FUNCTION_BLOCK CalibrationBlock
VAR_INPUT

	fbMotorReference : REFERENCE TO FB_AnalogMotorDriver; 	

END_VAR
VAR_OUTPUT

	// Variables for logging 
	nEncoder1Counts : LINT; 
	rEncoder1Degrees : REAL; 	
	
	// Variables for motor control 
	rCommand : REAL; 
	
	// Variables for load cell 
	rGripForce : REAL; 

END_VAR

// Constants used for the program 
VAR CONSTANT
	nMaxTrialNumber : UINT := 10; 
END_VAR

VAR
	
	// Variables to keep track of the actual encoder/motor setup
	fbEncoder1 : FB_QuadratureEncoder; 
	fbLoadCell : FB_AnalogLoadCellInput; // TODO: Change everything to top level reference maybe? 
	
	////// BEGIN GUI TEST OPTIONS
	//// All fields in the next section are in some way or another set by the GUI, and define 
	//// the type of test to take place.
	// 1. Test type
	bTestTypeHuman : BOOL; // Whether or not this a human or motor test 
	bTestTypeHumanLIVE : BOOL; 
	
	// 2. Number of trials
	nTrialNumber : UINT := 1; // Number of calibration trials to run in succession 
	nTrialNumberLIVE : UINT; 
	
	// 3. Trigger type
	bManualPulse : BOOL; // Whether to use manual pulse or grip schedule. 
	bManualPulseLIVE : BOOL; 
	bManualPulseTimerEnable : BOOL; 
	bManualPulseTimerEnableLIVE : BOOL;
	rManualPulseTimerValue : REAL; 
	rManualPulseTimerValueLIVE : REAL;
	
	// 4. Trigger controls
	bUseConstantGripTrigger : BOOL;
	bUseConstantGripTriggerLIVE : BOOL;
	aGripSchedule : ARRAY[1..nMaxTrialNumber] OF REAL;
	aGripScheduleLIVE : ARRAY[1..nMaxTrialNumber] OF REAL;  
	rCurrentGripThreshold : REAL := 0; 
	
	// 5. Pulse controls 
	bUseConstantPulseTorque : BOOL; 
	bUseConstantPulseTorqueLIVE : BOOL;
	rConstantTorqueSetting : REAL; 	
	rConstantTorqueSettingLIVE : REAL;

	// 6. Test Controls
	bLaunchTestSequence : BOOL := FALSE; // Triggers an entry into the testing loop. 
 
	/////// END GUI TEST OPTIONS
	
	// State machine for actual calibration logic. 
	// At the begginning, we are in the configuration state. 
	eSequenceState : CalibStateType := CalibStateType.PRE_LAUNCH; 
	eNextSequenceState : CalibStateType := CalibStateType.PRE_LAUNCH; 
	nCurrentTestIndex : INT := 0; 
	bTestIsLive : BOOL := FALSE; 
	bTestIsLiveTrigger : BOOL := FALSE; 
	
	// Helper variables 
	i : UINT; 
	fbTonTest : TON := (PT := T#1000MS); // Timer for the entire test
	fbTonPulse : TON := (PT := T#200MS); // Timer for the duration of the pulse 
	bMotorLimitHit : BOOL := FALSE; 

END_VAR

///////////// Read sensors on current iteration
// Encoders 
fbEncoder1(); 
nEncoder1Counts := fbEncoder1.nNetCounts; 
rEncoder1Degrees := fbEncoder1.rDegrees; 

// Load cell 
fbLoadCell(); 
rGripForce := fbLoadCell.rCalibratedOutput; 
///////////// End sensor reading 


// Update Timers 
// First we compute the timer update 
fbTonTest(IN := bTestIsLive); 
fbTonPulse(IN := bTestIsLive); 

// Now we go through the calibration logic. 
CASE eSequenceState OF
	
	// The user is currently setting permissions, we can update them live. 
	CalibStateType.PRE_LAUNCH:
	
		// First we start by updating options to the LIVE variables. 
		bTestTypeHumanLIVE := bTestTypeHuman; 
		nTrialNumberLIVE := nTrialNumber; 
		bManualPulseLIVE := bManualPulse; 
		bManualPulseTimerEnableLIVE := bManualPulseTimerEnable; 
		rManualPulseTimerValueLIVE := rManualPulseTimerValue;
		bUseConstantGripTriggerLIVE := bUseConstantGripTrigger; 
		
		FOR i := 1 TO nMaxTrialNumber DO
			aGripScheduleLIVE[i] := aGripSchedule[i]; 
		END_FOR
		
		bUseConstantPulseTorqueLIVE := bUseConstantPulseTorque;
		rConstantTorqueSettingLIVE := rConstantTorqueSetting; 
		
		IF bLaunchTestSequence THEN
			eNextSequenceState := CalibStateType.TEST_SETUP; 
			// Also set the first test index 
			nCurrentTestIndex := 1; 
			// And put this signal back down 
			bLaunchTestSequence := FALSE; 
		ELSE
			eNextSequenceState := CalibStateType.PRE_LAUNCH; 
		END_IF
		
		// We also need to make sure any motor commands are no longer hanging over 
		bTestIsLive := FALSE; 
		rCommand := 0; 
		fbMotorReference(rCommandVoltage := rCommand); 
		
	// We are getting the test ready. 
	CalibStateType.TEST_SETUP: 
	
		// In this state, we need to recenter the motor back to the 0 point, and we also need to wait 
		// for the triggering signal. This signal is either going to be a timer, a manual button, or a grip threshold. 
		// We need to additionally resolve this for the test to commence. 
		
		// Reset motor limit flag if its been hit 
		bMotorLimitHit := FALSE; 
		
		// We can start by returning the motor to the homing position, which we can do with a simple PID
		rCommand := -1 * 3 * ((3/2) * (fbEncoder1.rDegrees / 90) - (1/2) * (fbEncoder1.rLastDegrees / 90));
		fbMotorReference(rCommandVoltage := rCommand); 
		
		// Then we check to see if the test going live conditions are met: 
		// We need to figure out the type of trigger that's being used, and then we test for that. 
		// In the first scenario, it's if there is a manual pulse sent from the button
		IF bTestIsLiveTrigger AND bManualPulseLIVE AND NOT bManualPulseTimerEnableLIVE THEN // Manually push button 
			bTestIsLive := TRUE; 
			bTestIsLiveTrigger := FALSE; 
		END_IF 
		
		// Then we need to check if it's a grip trigger pulse. To do this, we first update what the grip trigger
		// should be, and then we check to see if the current grip matches that value 
		IF NOT bManualPulseLIVE THEN
			IF bUseConstantGripTrigger THEN
				rCurrentGripThreshold := aGripScheduleLIVE[1]; 
			ELSE
				rCurrentGripThreshold := aGripScheduleLIVE[nCurrentTestIndex]; 
			END_IF
			
			// Once we've set the value, we can compare to see if we've reached it 
			IF rGripForce > rCurrentGripThreshold THEN
				bTestIsLive := TRUE; 
			END_IF
			
		END_IF
		
		IF bTestIsLive THEN
			eNextSequenceState := CalibStateType.TEST_ACTIVE; 
		END_IF
		
		
	// Then we handle logic for actually completing the test. 
	CalibStateType.TEST_ACTIVE: 
	
		// Timer is set based on bTestIsLive variable. Timers are updated at the beginning of every cycle. 	
		IF NOT fbTonPulse.Q THEN // If the pulse hasn't expired, send the pulse 
			rCommand := MotorTorqueToCommandV(rCommandTorque := rConstantTorqueSettingLIVE); 
		ELSE
			rCommand := 0;
		END_IF
		
		// Check to see if motor has hit limit
		IF rEncoder1Degrees > 120 OR bMotorLimitHit THEN // hardcoded threshold, reset back to normal
			bMotorLimitHit := TRUE; 
			rCommand := -1 * 1.5 * ((3/2) * (fbEncoder1.rDegrees / 120) - (1/2) * (fbEncoder1.rLastDegrees / 120));
		END_IF
		
		fbMotorReference(rCommandVoltage := rCommand); 
	
		IF fbTonTest.Q THEN
			IF nCurrentTestIndex < UINT_TO_INT(nTrialNumberLIVE) THEN // We have more tests to run 
				bTestIsLive := FALSE;
				nCurrentTestIndex := nCurrentTestIndex + 1; 
				eNextSequenceState := CalibStateType.TEST_SETUP;
			ELSE	
				eNextSequenceState := CalibStateType.TEST_FINISHED; 
				bTestIsLive := FALSE; 
			END_IF
				
		END_IF

END_CASE

// Update everything that just happened and log the event. 


// Update state for next iteration
eSequenceState := eNextSequenceState; 

GVL.ENCODER_1_COUNTER_VALUE := nEncoder1Counts; 
GVL.ENCODER_1_DEGREES := rEncoder1Degrees; 
GVL.MOTOR_1_APPLIED_VOLTAGE := rCommand;
GVL.LOAD_CELL_NEWTONS := rGripForce;

METHOD Reset : BOOL
VAR_INPUT
END_VAR
fbEncoder1.Reset();
END_METHOD

END_FUNCTION_BLOCK

(* stored: Version 1.1.0.1, ProductVersion 3.1.4024.12
   POU CalibrationBlock: Id {808fb392-0321-4ad3-ac5f-7deb84640061}, SpecialFunc None
   Method Reset: Id {3efb2b45-adfc-4639-850c-d3b8867d9734} *)
